(* IEC 61131-3 sources: Std_PalletMover/Class/MainLedControl, 1 file *)

(* ---- MainLedControl.st ---- *)
(*!
<Class
	Name               = "MainLedControl"
	Revision           = "0.0"
	RealtimeTask       = "false"
	CyclicTask         = "false"
	BackgroundTask     = "false"
	Sigmatek           = "false"
	OSInterface        = "false"
	HighPriority       = "false"
	Automatic          = "false"
	UpdateMode         = "Prescan"
	SharedCommandTable = "true"
	Objectsize         = "(1020,240)">
	<Channels>
		<Server Name="SetLeds" Visualized="false" Initialize="false" WriteProtected="false" Retentive="false"/>
		<Client Name="AgvConfig" Required="true" Internal="false"/>
		<Client Name="AgvSettings" Required="true" Internal="false"/>
		<Client Name="I_LedControl" Required="true" Internal="true"/>
		<Client Name="ToLedModule" Required="false" Internal="false"/>
	</Channels>
	<Network Name="MainLedControl">
		<!-- List of Components in this network -->
		<Components>
			<Object
				Name       = "_base"
				Class      = "PeripheralsBase"
				Position   = "(218,120)"
				Visualized = "false">
				<Channels>
					<Server Name="ObjectStatus"/>
					<Server Name="ToObject"/>
					<Client Name="op_LogData"/>
					<Client Name="p_NextObject"/>
				</Channels>
			</Object>
			<Object
				Name       = "I_LedControl"
				Class      = "I_LedControl"
				Position   = "(210,360)"
				Visualized = "false">
				<Channels>
					<Server Name="ClassSvr"/>
					<Server Name="SetLeds"/>
				</Channels>
			</Object>
		</Components>
		<Comments>
		</Comments>
		<!-- List of Connections in this network -->
		<Connections>
			<Connection Source="this.ToObject" Destination="_base.ToObject" Vertices="(976,210),(804,210),"/>
			<Connection Source="_base.op_LogData" Destination="this.op_LogData" Vertices="(218,210),(38,210),"/>
			<Connection Source="_base.p_NextObject" Destination="this.p_NextObject" Vertices="(218,270),(38,270),"/>
			<Connection Source="this.I_LedControl" Destination="I_LedControl.ClassSvr"/>
			<Connection Source="this.ObjectStatus" Destination="_base.ObjectStatus" Vertices="(976,270),(804,270),"/>
			<Connection Source="this.SetLeds" Destination="I_LedControl.SetLeds" Vertices="(976,330),(796,510),"/>
		</Connections>
		<!-- Headerfiles -->
		<Options>
		</Options>
	</Network>
</Class>
*)
#pragma using PeripheralsBase

MainLedControl : CLASS
: PeripheralsBase
  //Servers:
	SetLeds 	: SvrCh_LedState_PTofCls_I_LedControl;
  //Clients:
	ToLedModule 	: CltChCmd_PL221;
	I_LedControl 	: CltChCmd_I_LedControl;
	AgvConfig 	: CltChCmd_AgvConfig;
	AgvSettings 	: CltChCmd_AgvSettings;
  //Variables:
		SetCurrendEndLedState 	: DINT;
		ConfigStepper 	: DINT;
		StartUpStepper 	: DINT;
  //Functions:

	FUNCTION VIRTUAL GLOBAL HandleOperational
		VAR_OUTPUT
			RetValue 	: DINT;
		END_VAR;

	FUNCTION VIRTUAL GLOBAL Handleconfiguration
		VAR_OUTPUT
			RetValue 	: DINT;
		END_VAR;

	FUNCTION VIRTUAL GLOBAL HandleStartUp
		VAR_OUTPUT
			RetValue 	: DINT;
		END_VAR;

	FUNCTION GetConfig;

	FUNCTION GetSettings;

	FUNCTION VIRTUAL GLOBAL SetLeds::Read
		VAR_OUTPUT
			output (EAX) 	: I_LedControl::LedState;
		END_VAR;

	FUNCTION VIRTUAL GLOBAL SetLeds::Write
		VAR_INPUT
			input (EAX) 	: I_LedControl::LedState;
		END_VAR
		VAR_OUTPUT
			result (EAX) 	: I_LedControl::LedState;
		END_VAR;
  //Tables:
	FUNCTION @STD
		VAR_OUTPUT
			ret_code	: CONFSTATES;
		END_VAR;
	FUNCTION GLOBAL TAB @CT_;
END_CLASS;

#pragma using I_LedControl
#pragma usingLtd AgvConfig
#pragma usingLtd AgvSettings
#pragma usingLtd PL221

FUNCTION VIRTUAL GLOBAL MainLedControl::SetLeds::Read
	VAR_OUTPUT
		output (EAX) 	: I_LedControl::LedState;
	END_VAR

	SetLeds := I_LedControl.SetLeds.Read();
	output := SetLeds;

END_FUNCTION

FUNCTION VIRTUAL GLOBAL MainLedControl::SetLeds::Write
	VAR_INPUT
		input (EAX) 	: I_LedControl::LedState;
	END_VAR
	VAR_OUTPUT
		result (EAX) 	: I_LedControl::LedState;
	END_VAR

    SetLeds := input;
    result := SetLeds;

END_FUNCTION

FUNCTION VIRTUAL GLOBAL MainLedControl::Handleconfiguration
	VAR_OUTPUT
		RetValue 	: DINT;
	END_VAR

    case ConfigStepper of

        0:
                GetConfig();
                ConfigStepper += 1;
        1:

               RetValue := true;
      end_case;

END_FUNCTION

FUNCTION MainLedControl::GetConfig
// Use sensor and make connection with hardware

if AgvConfig.GetBooleanValue(Path:="AGV.Peripherals.BasicLedPl221.Connection.EnableObj") = true then
    ConnectClientChannels(AgvConfig.GetStringValue(Path:="AGV.Peripherals.BasicLedPl221.Connection.ToPlModule"));

end_if;

END_FUNCTION

FUNCTION VIRTUAL GLOBAL MainLedControl::HandleStartUp
	VAR_OUTPUT
		RetValue 	: DINT;
	END_VAR

    case StartUpStepper of

        0:
            GetSettings();
            StartUpStepper += 1;
         1:

            StartUpStepper += 1;
         2:
            RetValue := true;

      end_case;

END_FUNCTION

FUNCTION VIRTUAL GLOBAL MainLedControl::HandleOperational
	VAR_OUTPUT
		RetValue 	: DINT;
	END_VAR

    case  I_LedControl.SetLeds of

        I_LedControl::LedState::LedAllOff:

        I_LedControl::LedState::LedRed:

        I_LedControl::LedState::LedRedLeft:

        I_LedControl::LedState::LedRedRight:

        I_LedControl::LedState::LedGreen:

        I_LedControl::LedState::LedGreenLeft:

        I_LedControl::LedState::LedGreenRight:

        I_LedControl::LedState::LedBlue:

        I_LedControl::LedState::LedBlueLeft:

        I_LedControl::LedState::LedBlueRight:

      end_case;

END_FUNCTION

FUNCTION MainLedControl::GetSettings

END_FUNCTION
